// ---- Tests/TcoSequenceObserver/TcoSequenceObserverTests.TcPOU
FUNCTION_BLOCK TcoSequenceObserverTests EXTENDS TcoCore._internals_TcoContext
VAR
    _s : TcoCore.TcoSequence(THIS^, eRestoreMode.None);
    _sObserver : TcoCore.TcoSequencerObserver(THIS^);
END_VAR

(*~
    <docu>
        <summary>
            Main method of the TcoContext. This is the entry point of any control logic that belongs to this context.
            The call of this method is ensured by calling the <c>InstanceName.Run()</c> method, and it must not be called explicitly.
            This method is abstract, and it must be overridden in derived block.
        </summary>
    </docu>
~*)
METHOD PROTECTED Main
CASE _testId OF
    eTcoSequenceObserverTests.RestoreSequencer:
        _s.Restore();
        _sObserver.Clear();
    eTcoSequenceObserverTests.RunSequenceWithObserverTest:
        RunSequencerWithObserver();
    eTcoSequenceObserverTests.RunSequenceWithoutObserverTest:
        RunSequencerWithoutObserver();
END_CASE
END_METHOD

METHOD RunSequencerWithObserver
VAR_INPUT
END_VAR
_s.Open();
THIS^._s.Observer := _sObserver;
THIS^._s.Messenger.Info('Stations two sequencer is running.');

IF (_s.Step(100, TRUE, '100')) THEN
    //-----------------------------------------------------
    _s.StepCompleteWhen(_s.CurrentStep.Duration >= T#10MS);
    //-----------------------------------------------------
END_IF

IF (_s.Step(200, TRUE, '200')) THEN
    //-----------------------------------------------------
    _s.StepCompleteWhen(_s.CurrentStep.Duration >= T#20MS);
    //-----------------------------------------------------
END_IF

IF (_s.Step(300, TRUE, '300')) THEN
    //-----------------------------------------------------
    _s.StepCompleteWhen(_s.CurrentStep.Duration >= T#30MS);
    //-----------------------------------------------------
END_IF

IF (_s.Step(400, TRUE, '400')) THEN
    //-----------------------------------------------------
    _s.StepCompleteWhen(_s.CurrentStep.Duration >= T#40MS);
    //-----------------------------------------------------
END_IF

IF (_s.Step(500, TRUE, '500')) THEN
    //-----------------------------------------------------
    THIS^.ProbeDoneWhen(TRUE);
    _s.Restore();
    //-----------------------------------------------------
END_IF

_s.Close();
END_METHOD

METHOD RunSequencerWithoutObserver
VAR_INPUT
END_VAR
_s.Open();
THIS^._s.Observer := 0;
THIS^._s.Messenger.Info('Stations two sequencer is running.');

IF (_s.Step(100, TRUE, '100')) THEN
    //-----------------------------------------------------
    _s.StepCompleteWhen(_s.CurrentStep.Duration >= T#250MS);
    //-----------------------------------------------------
END_IF

IF (_s.Step(200, TRUE, '200')) THEN
    //-----------------------------------------------------
    _s.StepCompleteWhen(_s.CurrentStep.Duration >= T#100MS);
    //-----------------------------------------------------
END_IF

IF (_s.Step(300, TRUE, '300')) THEN
    //-----------------------------------------------------
    _s.StepCompleteWhen(_s.CurrentStep.Duration >= T#50MS);
    //-----------------------------------------------------
END_IF

IF (_s.Step(400, TRUE, '400')) THEN
    //-----------------------------------------------------
    _s.StepCompleteWhen(_s.CurrentStep.Duration >= T#25MS);
    //-----------------------------------------------------
END_IF

IF (_s.Step(500, TRUE, '500')) THEN
    //-----------------------------------------------------
    THIS^.ProbeDoneWhen(TRUE);
    _s.Restore();
    //-----------------------------------------------------
END_IF

_s.Close();
END_METHOD

END_FUNCTION_BLOCK

// ---- Components/fbPiston.TcPOU
{attribute addProperty Name "Pneumatic cyclinder"}
FUNCTION_BLOCK fbPiston EXTENDS TcoCore.TcoComponent IMPLEMENTS IPistonGripper, IPistonHorizontal, IPistonVertical
VAR_INPUT
    iHomePositionSensor : BOOL;
    iWorkPositionSensor : BOOL;
END_VAR
VAR_OUTPUT
    qHomePositionActuator : BOOL;
    qWorkPositionActuator : BOOL;
END_VAR
VAR
    {attribute addProperty Activity "moves to home position"}
    _moveHomeTask : fbPistonMoveTask(THIS^);
    {attribute addProperty Activity "moves to work position"}
    _moveWorkTask : fbPistonMoveTask(THIS^);
    _moveHomeMomentaryTask : TcoCore.TcoMomentaryTask(THIS^);
    _moveHomeToggleTask : TcoCore.TcoToggleTask(THIS^, FALSE);
    _config : fbPistonConfig;
    _status : fbPistonStatus;
END_VAR

_moveHomeTask(PositionSensor := iHomePositionSensor, MoveToPositionSignal := qHomePositionActuator, InverseSignal := qWorkPositionActuator);
_moveWorkTask(PositionSensor := iWorkPositionSensor, MoveToPositionSignal := qWorkPositionActuator, InverseSignal := qHomePositionActuator);
_moveHomeMomentaryTask.Run();
_moveHomeToggleTask.Toggle();

METHOD Close : TcoCore.ITcoTaskStatus
Close := MoveToHome();
END_METHOD

METHOD MoveDown : TcoCore.ITcoTaskStatus
MoveDown := MoveToHome();
END_METHOD

METHOD MoveLeft : TcoCore.ITcoTaskStatus
MoveLeft := MoveToWork();
END_METHOD

METHOD MoveRight : TcoCore.ITcoTaskStatus
MoveRight := MoveToHome();
END_METHOD

METHOD PROTECTED MoveToHome : TcoCore.ITcoTaskStatus
MoveToHome := THIS^._moveHomeTask.Invoke();
END_METHOD

METHOD PROTECTED MoveToWork : TcoCore.ITcoTaskStatus
MoveToWork := THIS^._moveWorkTask.Invoke();
END_METHOD

METHOD MoveUp : TcoCore.ITcoTaskStatus
MoveUp := MoveToWork();
END_METHOD

METHOD Open : TcoCore.ITcoTaskStatus
Open := MoveToWork();
END_METHOD

METHOD Restore : ITcoRestorable
THIS^._moveHomeTask.Restore();
THIS^._moveWorkTask.Restore();
END_METHOD

(*~
    <docu>
        <summary>
            Custom service (manual, maintenance) logic.
            This method must be implemented in derived class.
        </summary>
    </docu>
~*)
METHOD PROTECTED ServiceMode
END_METHOD

END_FUNCTION_BLOCK

// ---- Components/fbPistonMoveTask.TcPOU
{attribute addProperty Activity "task is running"}
FUNCTION_BLOCK fbPistonMoveTask EXTENDS TcoCore.TcoTask
VAR_INPUT
    PositionSensor : BOOL;
END_VAR
VAR_IN_OUT
    MoveToPositionSignal : BOOL;
    InverseSignal : BOOL;
END_VAR

IF (THIS^.Execute()) THEN
    THIS^.Messenger.Debug('|[[1]AttributeName]| |[AttributeActivity]|, extremity sensor not reached yet.');
    InverseSignal := FALSE;
    MoveToPositionSignal := TRUE;
    ThrowWhen(THIS^.ElapsedTime > T#5S);
    THIS^.DoneWhen(PositionSensor);
END_IF

END_FUNCTION_BLOCK

// ---- Tests/TcoSequence/PlcExecuted/TcoSequenceTestChildState.TcPOU
FUNCTION_BLOCK TcoSequenceTestChildState EXTENDS TcoCore.TcoState
VAR
    _requestedState : UINT;
    _requestedStateCount : ULINT;
    _restoreCount : ULINT;
END_VAR

(*~
    <docu>
        <summary>
            This method is called on each change of the <c>State</c>. This method could be overloaded and custom code should be placed here.
        </summary>
    </docu>
~*)
METHOD PROTECTED OnStateChange
VAR_INPUT
    PreviousState : INT;
    NewState : INT;
END_VAR
IF NewState = _requestedState THEN
    _requestedStateCount := _requestedStateCount + 1;
END_IF

IF NewState = -1 THEN
    _restoreCount := _restoreCount + 1;
END_IF
END_METHOD

PROPERTY RequestedState : UINT
GET
RequestedState := _requestedState;
END_GET
SET
_requestedState := RequestedState;
END_SET
END_PROPERTY

END_FUNCTION_BLOCK
